Fanuc KAREL source: kf00101.KL

-- PROVISIONAL review KL for V770-1; original PC SHA256 611aeb3c245198c9dca64d0bdd0a9db9f6c5ca304298818d26703e26a687f0ac
-- Incomplete behavior may be omitted. Consult companion uncertainty JSON. Do not deploy.
PROGRAM KF00101
%NOLOCKGROUP
BEGIN
  -- UNRESOLVED_PC offsets 5-16; opcodes 2E,23
  -- UNRESOLVED_PC offsets 21-32; opcodes 2E,23
  -- UNRESOLVED_PC offsets 37-63; opcodes 27,27,9D,22,27,9D,31,7E,4A
  -- UNRESOLVED_PC offsets 68-72; opcodes 7F
END KF00101
